PROGRAM Temperatur
VAR
END_VAR

CASE SM.Status OF
	
	Lesen:
	
		Temp_VD_in.REAL_VAR			:= FB_SPS_zu_Nativ_lin 		(Input := Temp_VD_in);
		Temp_VD_out.REAL_VAR		:= FB_SPS_zu_Nativ_lin 		(Input := Temp_VD_out);
		
		Temp_VD_in_rev.REAL_VAR		:= FB_SPS_zu_Nativ_lin 		(Input := Temp_VD_in_rev);
		Temp_VD_out_rev.REAL_VAR	:= FB_SPS_zu_Nativ_lin 		(Input := Temp_VD_out_rev);
		
		Temp_VD_surface1.REAL_VAR	:= FB_SPS_zu_Nativ_lin 		(Input := Temp_VD_surface1);
		Temp_VD_surface2.REAL_VAR	:= FB_SPS_zu_Nativ_lin 		(Input := Temp_VD_surface2);
		Temp_VD_surface3.REAL_VAR	:= FB_SPS_zu_Nativ_lin 		(Input := Temp_VD_surface3);
		Temp_VD_surface4.REAL_VAR	:= FB_SPS_zu_Nativ_lin 		(Input := Temp_VD_surface4);
		Temp_VD_surface5.REAL_VAR	:= FB_SPS_zu_Nativ_lin 		(Input := Temp_VD_surface5);
		Temp_VD_surface6.REAL_VAR	:= FB_SPS_zu_Nativ_lin 		(Input := Temp_VD_surface6);
				
		Temp_VF_in.REAL_VAR			:= FB_SPS_zu_Nativ_lin 		(Input := Temp_VF_in);
		Temp_VF_out.REAL_VAR		:= FB_SPS_zu_Nativ_lin 		(Input := Temp_VF_out);
		
		Temp_VD_defrost_in.REAL_VAR	:= FB_SPS_zu_Nativ_lin	 	(Input := Temp_VD_defrost_in);
		Temp_VD_defrost_out.REAL_VAR:= FB_SPS_zu_Nativ_lin 		(Input := Temp_VD_defrost_out);

		Temp_KP_in.REAL_VAR			:= FB_SPS_zu_Nativ_lin 		(Input := Temp_KP_in);
		Temp_KP_out.REAL_VAR		:= FB_SPS_zu_Nativ_lin 		(Input := Temp_KP_out);
		
		Temp_vor_EV.REAL_VAR		:= FB_SPS_zu_Nativ_lin 		(Input := Temp_vor_EV);
		Temp_vor_EV_rev.REAL_VAR	:= FB_SPS_zu_Nativ_lin 		(Input := Temp_vor_EV_rev);
	
		(*Gemittelte Temperatur auf der Oberflächentemperatur auf dem Verdampfer*)
	Temp_VD_Surface_gemittelt := 0.25*(Temp_VD_surface6.REAL_VAR+Temp_VD_surface5.REAL_VAR+Temp_VD_surface4.REAL_VAR+Temp_VD_surface2.REAL_VAR);
	

	

	
	Schreiben:
		//kein Schreiben notwendig

END_CASE

END_PROGRAM

(* stored: Version 1.1.0.1, ProductVersion 3.1.4019.2
   POU Temperatur: Id {4d77f1ad-8412-447f-bda7-dbbf6e6d3ab0}, SpecialFunc None *)
